RESOURCE_TYPE Config_EMB_RES (* Basic resource with configuration inputs *)
  (* Function: This resource is based on the basic resource for executing FB networks with the additional functionality of configuration data inputs. It already contains an instance of the E_RESTART FB providing events for starting up and shutting down an application.  This resource is based on examples found in the different parts of IEC 61499 and the documentation at http://www.holobloc.com/doc/fb/rt/EMB_RES.htm; Description: Copyright (c) 2024 Primetals Technologies Austria GmbH This program and the accompanying materials are made available under the terms of the Eclipse Public License 2.0 which is available at https://www.eclipse.org/legal/epl-2.0/ SPDX-License-Identifier: EPL-2.0 *)
  (* Version 3.0, 2025-04-14, Patrick Aigner, changed package *)
  (* Version 1.0, 2024-04-02, Markus Meingast, Primetals Technologies Austria GmbH *)
  PACKAGE iec61499::system;
  VAR_INPUT
    OPCUA_Namespace : WSTRING; (* OPC UA Namespace *)
  END_VAR
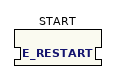
  FBS
    START : iec61499::events::E_RESTART;
  END_FBS
END_RESOURCE_TYPE
